(* Schneider Machine Expert - Basic project EX04, file version 1.8.0.0 *)
(* ProjectInformations: Name=New project *)

HARDWARE
  Cpu 0: TM221CE16R
  EthernetConfiguration: NetworkName=M221, IpAllocationMode=FixedAddress, IpAddress=192.168.162.202, SubnetMask=255.255.255.0
  SerialLineConfiguration: Baud=Baud19200, Parity=ParityEven, DataBits=DataBits8, StopBits=StopBits1, PhysicalMedium=PhysicalMediumRs485, TransmissionMode=TransmissionModeModbusRtu, SlaveId=1, Addressing=SlaveAddressing
  MastTask: UsePeriodScanMode=false, PeriodScan=100
  FastTask: Period=255
  CpuBehavior: StartingMode=StartAsPreviousState, AutoSaveRamOnEeprom=true, WatchdogPeriod=250

SYMBOLS  (address, symbol, comment, settings)

POU New POU
  (* SectionNumber=1 *)

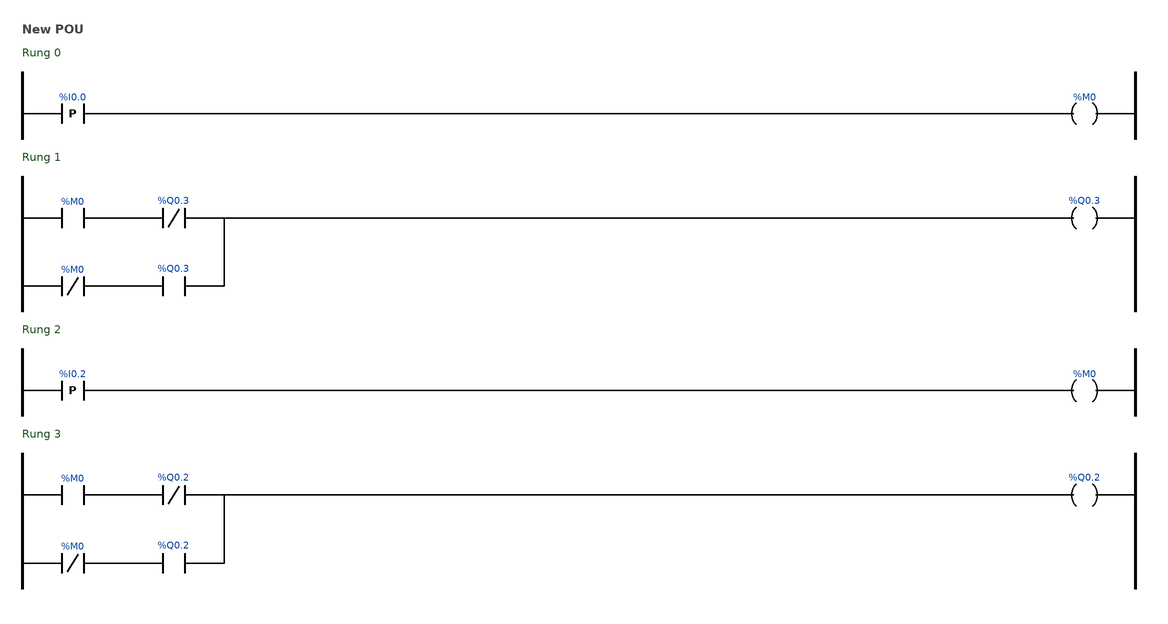

// Rung 0
  LDR %I0.0
  ST %M0
  // as ST:
  //   %M0 := RISING(%I0.0);

// Rung 1
  LD %M0
  ANDN %Q0.3
  OR(N %M0
  AND %Q0.3
  )
  ST %Q0.3
  // as ST:
  //   %Q0.3 := %M0 AND NOT %Q0.3 OR NOT %M0 AND %Q0.3;

// Rung 2
  LDR %I0.2
  ST %M0
  // as ST:
  //   %M0 := RISING(%I0.2);

// Rung 3
  LD %M0
  ANDN %Q0.2
  OR(N %M0
  AND %Q0.2
  )
  ST %Q0.2
  // as ST:
  //   %Q0.2 := %M0 AND NOT %Q0.2 OR NOT %M0 AND %Q0.2;
